PROGRAM SIMULATOR
VAR
	ship1 : ShipSimulator(0);
	ship2 : ShipSimulator(20);
END_VAR


ship1();

ship2();

END_PROGRAM

(* stored: Version 1.1.0.1, ProductVersion 3.1.4020.12
   POU SIMULATOR: Id {b537270b-d5b9-4044-8e1f-03b2cd92e219}, SpecialFunc None *)
